// TIA Portal V18 export
FUNCTION_BLOCK "LightBarrier"   // FB75, FBD
{ S7_Optimized_Access := 'TRUE' }
VERSION : 0.1
// stored: AutoNumber true, IsIECCheckEnabled false, IsRetainMemResEnabled false, MemoryReserve 100, SetENOAutomatically false, UDAEnableTagReadback false
   VAR_INPUT
      barrier_ok : Bool;
   END_VAR
BEGIN
END_FUNCTION_BLOCK
